// TIA Portal V17 export
// export: Created 2024-08-07T21:44:14.669822Z, ExportSetting WithDefaults, DisplayName Totally Integrated Automation Portal, DisplayVersion V17 Update 7, DisplayName TIA Portal Openness, DisplayVersion V17 Update 7, DisplayName TIA Portal Version Control Interface, DisplayVersion V17, DisplayName SINAMICS Startdrive Advanced, DisplayVersion V17 SP2, DisplayName SINAMICS Startdrive G110M, G120, G120C, G120D, G120P, G115D, DisplayVersion V17 SP2, DisplayName SINAMICS Startdrive G130, G150, S120, S150, SINAMICS MV, S210, DisplayVersion V17 SP2, DisplayName STEP 7 Professional, DisplayVersion V17 Update 7, DisplayName STEP 7 Safety, DisplayVersion V17 Update 6, DisplayName WinCC Advanced / Unified PC, DisplayVersion V17 Update 7
TYPE "UDT_Digiforce"
// stored: IsFailsafeCompliant false
   STRUCT
      programActual : USInt;
      programOK : Bool;
      ProgramChangeNOK : Bool;
      programSet : USInt;
      ActualWay : Real;
      ActualForce : Real;
      Ready : Bool;
      ResultOK : Bool;
      ResultNOK : Bool;
      Auto : Bool;
      Start : Bool;
      Running : Bool;
      TareX : Bool;
   END_STRUCT;
END_TYPE
